PROGRAM PROP_MAIN
VAR
	barcodeState : E_Barcode_State := E_Barcode_State.INIT;
	newData : BYTE := 16#00;
	
	positionValues_Front : ARRAY[0..3] OF BYTE;
	velocityValues_Front : ARRAY[0..1] OF BYTE; 
	
	positionValues_Back : ARRAY[0..3] OF BYTE;
	velocityValues_Back : ARRAY[0..1] OF BYTE; 
	
	position_Front : DINT;
	velocity_Front : DINT;
	
	position_Back : DINT;
	velocity_Back : DINT;
	
	positionDelft_Front : DINT;
	positionDelft_Back	: DINT;
	
	quality : INT;
	
	start : BOOL := FALSE;
	
	Send_CAN_Command : FB_SendPosVelocity;
	Receive_CAN_Current : FB_ReceiveCurrent;
	Receive_CAN_Temp : FB_ReceiveTemp;
	
	Id_ref : LREAL;
	Iq_ref : LREAL;
	Id_filtered : LREAL;
	Iq_filtered : LREAL;
	
	Temp_a_gd : LREAL;
	Temp_b_gd : LREAL;
	Temp_c_gd : LREAL;
	
	delft_converter : FB_PositionConverter;
END_VAR

VAR CONSTANT
	SCALE_FACTOR : INT := 100;
	BARCODE_START : INT := 11920;
	SET_COMMAND : BYTE := 16#01;
	SEND_POS_VEL : BYTE := 16#80;
	SEND_DIAG : BYTE := 16#08;
	SEND_MARKER_INFO : BYTE := 16#02;
	OFFSET_FRONT	: DINT;
	OFFSET_BACK		: DINT;
END_VAR

CASE barcodeState OF
	
	E_Barcode_State.INIT:
	
		IF start THEN
			barcodeState := E_BARCODE_STATE.SEND_POS_VEL_COMMAND;
		END_IF
		
	E_Barcode_State.SEND_POS_VEL_COMMAND:
		
		positionValues_Front[0] := GVL_PROP.InputData1_Front[4];
		positionValues_Front[1] := GVL_PROP.InputData1_Front[5];
		positionValues_Front[2] := GVL_PROP.InputData1_Front[6];
		positionValues_Front[3] := GVL_PROP.InputData1_Front[7];
		
		velocityValues_Front[0] := GVL_PROP.InputData2_Front[0];
		velocityValues_Front[1] := GVL_PROP.InputData2_Front[1];
		
		IF velocityValues_Front[0] > 128 THEN
			velocity_Front := (256 * 256 - (256 * velocityValues_Front[0] + velocityValues_Front[1]));
		ELSE
			velocity_Front := 256 * velocityValues_Front[0] + velocityValues_Front[1];	
		END_IF
		
		position_Front := 
			256 * 256 * 256 * positionValues_Front[0]
			+ 256 * 256 * positionValues_Front[1]
			+ 256 * positionValues_Front[2]
			+ positionValues_Front[3];
			
		delft_converter(diReadValue := position_Front, diPosition => positionDelft_Front);
		
		position_Front := position_Front / SCALE_FACTOR - BARCODE_START;
		
		newData := newData XOR 16#80; // -> only toggled once every cycle since the the newdata toggled is shared between the two 
		
		GVL_PROP.OutputData_Front[0] := newData OR SET_COMMAND;
		GVL_PROP.OutputData_Front[2] := SEND_POS_VEL;
		
		//-------------------------------------------

		positionValues_Back[0] := GVL_PROP.InputData1_Front[4];
		positionValues_Back[1] := GVL_PROP.InputData1_Front[5];
		positionValues_Back[2] := GVL_PROP.InputData1_Front[6];
		positionValues_Back[3] := GVL_PROP.InputData1_Front[7];
		
		velocityValues_Back[0] := GVL_PROP.InputData2_Back[0];
		velocityValues_Back[1] := GVL_PROP.InputData2_Back[1];
		
		IF velocityValues_Back[0] > 128 THEN
			velocity_Back := (256 * 256 - (256 * velocityValues_Back[0] + velocityValues_Back[1]));
		ELSE
			velocity_Back := 256 * velocityValues_Back[0] + velocityValues_Back[1];	
		END_IF
		
		position_Back := 
			256 * 256 * 256 * positionValues_Back[0]
			+ 256 * 256 * positionValues_Back[1]
			+ 256 * positionValues_Back[2]
			+ positionValues_Back[3];
			
		delft_converter(diReadValue := position_Back, diPosition => positionDelft_Back);
			
		position_Back := position_Back / SCALE_FACTOR - BARCODE_START;;
		
		GVL_PROP.OutputData_Back[0] := newData OR SET_COMMAND;
		GVL_PROP.OutputData_Back[2] := SEND_POS_VEL;		
		
		
		
	E_Barcode_State.SEND_DIAGNOSTIC_COMMAND:
		newData := newData XOR 16#80;
		GVL_PROP.OutputData_Front[0] := newData OR SET_COMMAND;
		GVL_PROP.OutputData_Front[2] := 16#00;
		GVL_PROP.OutputData_Front[3] := SEND_DIAG;
		
	E_Barcode_State.SEND_MARKER_INFO_COMMAND:
		newData := newData XOR 16#80;
		GVL_PROP.OutputData_Front[0] := newData OR SET_COMMAND;
		GVL_PROP.OutputData_Front[2] := 16#00;
		GVL_PROP.OutputData_Front[3] := SEND_MARKER_INFO;
		
	E_Barcode_State.ERROR:
		barcodeState := E_Barcode_State.INIT;
		start := FALSE;
	
END_CASE

Send_CAN_Command(Position := position_Front,
	Velocity := velocity_Front, 
	CAN_OUTPUTS := GVL_PropCAN.CAN_OUTPUTS, 
	CAN_INPUTS := GVL_PropCAN.CAN_INPUTS);

Receive_CAN_Current(Inputs := GVL_PropCAN.CAN_INPUTS, 
	Outputs := GVL_PropCAN.CAN_OUTPUTS);
	
Id_ref := Receive_CAN_Current.Id_ref;
Iq_ref := Receive_CAN_Current.Iq_ref;
Id_filtered := Receive_CAN_Current.Id_filtered;
Iq_filtered := Receive_CAN_Current.Iq_filtered;	

Receive_CAN_Temp(Inputs := GVL_PropCAN.CAN_INPUTS, 
	Outputs := GVL_PropCAN.CAN_OUTPUTS);
	
Temp_a_gd := Receive_CAN_Temp.Temp_a_gd;
Temp_b_gd := Receive_CAN_Temp.Temp_b_gd;
Temp_c_gd := Receive_CAN_Temp.Temp_c_gd;

END_PROGRAM

(* stored: Version 1.1.0.1
   POU PROP_MAIN: Id {6203b0f5-9def-42aa-a1a3-50bbae11de91}, SpecialFunc None *)
